# EPICS substitutions: vacuum/MAIN_TRUNK/vacApp/Db/l406_agilent4uhv.substitutions
# Agilent4UHV substitutions file

file db/agilent4uhv.db
{
     pattern {LOCA,			DEV,			PORT,		ADDR,	TIMEOUT}
     		{HL4,			VL406_1,		4uhv_1,		0,		0.2}
     		{HL4,			VL406_2,		4uhv_2,		0,		0.2}
}

file db/agilent4uhv_alias.db
{
     pattern {LOCA,			DEV,			SUB1,				SUB2,				SUB3,					SUB4,				PORT,		ADDR,	TIMEOUT}
     		 {HL4,			VL406_1,		IP01:L406_Acc601,		IP02:L406_Acc602,		IP03:L406_Acc603,			IP04:L406_Acc604,		4uhv_1,		0,		0.2}
		 {HL4,			VL406_2,		IP05:L406_Acc605,		IP06:L406_Wave601,	IP07:L406_Kly601,			IP08:Empty,			4uhv_2,		0,		0.2}
}
